FUNCTION F_Sum : DINT;
VAR_IN_OUT
    aData     : ARRAY [*] OF DINT;
END_VAR
VAR
    i, nSum   : DINT;
END_VAR


nSum := 0;
FOR i := LOWER_BOUND(aData,1) TO UPPER_BOUND(aData,1) DO
    nSum := nSum + aData[i];
END_FOR;
F_Sum := nSum;

END_FUNCTION

(* stored: Version 1.1.0.1, ProductVersion 3.1.4024.12
   POU F_Sum: Id {0b785f83-0e8d-45a3-a633-da139c67b874}, SpecialFunc None *)
